# EPICS substitutions: ioc_manual/bsread.subs
file bsread.template {
	pattern{P} {BSREAD}
}
